FUNCTION_BLOCK FB_CalculateThicknessTestDouble IMPLEMENTS I_CalculateThickness
VAR
    fThickness : LREAL;
    nNumberOfTimesCalculateCalled : UINT;
END_VAR


METHOD Calculate
VAR_INPUT
    (* [1]*)
    fDesiredTransmission	: LREAL;
    (* [eV]*)
    fPhotonEnergy	: LREAL;
END_VAR
VAR_OUTPUT
    (* [mm]*)
    fThickness	: LREAL;
END_VAR

fThickness := THIS^.fThickness;

THIS^.nNumberOfTimesCalculateCalled := nNumberOfTimesCalculateCalled + 1;
END_METHOD


METHOD PUBLIC GetNumberOfTimesCalculateCalled : UINT

GetNumberOfTimesCalculateCalled := THIS^.nNumberOfTimesCalculateCalled;
END_METHOD


METHOD PUBLIC SetThickness
VAR_INPUT
    fThickness : LREAL;
END_VAR

THIS^.fThickness := fThickness;
END_METHOD

END_FUNCTION_BLOCK

(* stored: Version 1.1.0.1
   POU FB_CalculateThicknessTestDouble: Id {80820049-6f73-49ff-9ad0-7c5ccd408ffb}, SpecialFunc None
   Method Calculate: Id {786416ea-cfe9-41b5-b05f-de2a31b25ba7}
   Method GetNumberOfTimesCalculateCalled: Id {b4803615-8b00-4920-951d-83483299ed95}
   Method SetThickness: Id {c39c3097-3901-4c6f-919a-3966c6225d0c} *)
